# EPICS substitutions: db/Beckhoff_7XXX/ecmcEL7342.substitutions
file "ecmcEL7342-chX.template"
{
  pattern {CH_ID}
          {01   }
          {02   }
}

file "ecmcEL5101-chX.template"
{
  pattern {CH_ID}
          {01   }
          {02   }
}
